Fanuc KAREL source: ka00131.KL

-- PROVISIONAL review KL for V1013-1; original PC SHA256 d5f2b0a3b20868f066135ee4ab6104af56910053abf502229fca8b89f01513b9
-- Incomplete behavior may be omitted. Consult companion uncertainty JSON. Do not deploy.
PROGRAM KA00131
%NOLOCKGROUP
-- UNRESOLVED_DECL SRC type=002018
-- UNRESOLVED_DECL DST type=002018
BEGIN
  -- UNRESOLVED_PC offsets 5-19; opcodes 2E,22,9D,33,B2
  -- UNRESOLVED_PC offsets 24-42; opcodes 22,9D,33,B1,22,9D,33,B2
  -- UNRESOLVED_PC offsets 47-51; opcodes 7F
END KA00131
